Staubli VAL3: FILLSTR.pgx

program fillStr(string x_char, num x_num, string& x_return[])
  local num l_i
begin
  x_return=""
  if x_num>0
    for l_i=1 to x_num
      x_return=x_return+x_char
    endFor
  endIf
end
